// This function has been automatically generated from the project information.
{attribute 'signature_flag' := '1073741824'}
{attribute 'TcGenerated'}
{attribute 'no-analysis'}
FUNCTION F_GetTitle : WSTRING
VAR_INPUT
	
END_VAR

F_GetTitle := "CNM_CycleManagerInterfacesTests";

END_FUNCTION

(* stored: Version 1.1.0.1
   POU F_GetTitle: Id {90f0fdf2-31e1-42cc-8f21-752622ba7ec5}, SpecialFunc None *)
